TYPE ST_RV_Zustand :
STRUCT
	Betrieb_Anford			: BOOL;
	Betrieb_Soll			: BOOL;
	Betrieb					: BOOL;

	Stellung				: USINT;

	Regelung_Modus			: SINT;
	Regelung_Modus_wechsel  : BOOL;
	Regelung_Istw			: REAL;
	Regelung_Sollw_Anford	: REAL;
	Regelung_Sollw			: REAL;
	Regelung_Stellw			: REAL;

	Freigabe				: BOOL;
	Freigabe_Deakt			: BOOL;
	Freigabe_Code			: WORD;

	Stoerung				: BOOL;
	Stoerung_Code			: WORD;

	Warnung					: BOOL;
	Warnung_Code			: WORD;

	Status					: SINT;

	Status_Vorl				: BOOL;
	Status_Nachl			: BOOL;

	Quittierung				: BOOL;

END_STRUCT
END_TYPE

(* stored: Version 1.1.0.1, ProductVersion 3.1.4024.9
   DUT ST_RV_Zustand: Id {41e98ad4-1a25-4e1f-8cee-639e52e5d2cf} *)
